# EPICS substitutions: iocs/MC04/db/SAI_IOCsystem.substitutions
# DEVICE: device name
# CARD:
# CS_VERSION_VAL

file /opt/epics/modules/uIOCSystem/db/uIOCsystem.template {
pattern { DEVICE, CARD, CS_VERSION_VAL}
	{ "XF:06BMA-OP{MC:04}", "0", "v0.01" }
}

#EOF
